(* IEC 61131-3 sources: xPLCCore/codesys_code/Application/COMM_FBs/FB_MpPacker, 25 files *)

(* ---- FB_MpPacker.st ---- *)
FUNCTION_BLOCK FB_MpPacker
VAR_INPUT
END_VAR
VAR_OUTPUT
END_VAR
VAR
    // Builder-pattern slot binding. Caller invokes BindSlot(p) once per
    // reply/event acquisition (TryAcquireReplySlot / ProbeReplySlot /
    // TryAcquireReplySlotOrScratch on AxisGroupSM all auto-bind), then
    // the high-level KV/Pair/Elem helpers below use this stashed pointer
    // instead of taking the slot as a parameter at every call.
    //
    // Default 0 (NULL) -- a Pack* call before BindSlot will deref null
    // and crash deterministically; better than silently writing into
    // a stale slot. Re-bind on every acquire to make stale impossible.
    pSlot : POINTER TO MsgPakInfo := 0;
END_VAR
(* =========== IMPLEMENTATION =========== *)

(* ---- BindSlot.st ---- *)
METHOD BindSlot : BOOL
VAR_INPUT
    pBindSlot : POINTER TO MsgPakInfo;
END_VAR
(* =========== IMPLEMENTATION =========== *)
// Stash the active reply/event slot. All subsequent PackKv* / PackPair*
// / PackElem* / PackKvMap / PackKvArray calls target this slot until
// the next BindSlot. Called automatically by the AxisGroupSM slot-
// lifecycle helpers (TryAcquireReplySlot / ProbeReplySlot /
// TryAcquireReplySlotOrScratch); retry-style sites that hand-roll
// slot acquisition must call this themselves.
pSlot := pBindSlot;
BindSlot := TRUE;

(* ---- PackArrayHeader.st ---- *)
METHOD PackArrayHeader : POINTER TO BYTE
VAR_INPUT
	pStart : POINTER TO BYTE;
	uiCount : UINT;
END_VAR
VAR
	pWordCount : POINTER TO WORD;
END_VAR
(* =========== IMPLEMENTATION =========== *)
// Bound-slot guard (2026-10-04): if pStart lies in the slot bound by
// BindSlot and the up to 3 bytes would not fit, write nothing and flag the
// slot (the post-write checks of the PackKv* helpers only saw the
// overrun after the bytes were already in the next slot).
IF (pSlot <> 0) AND (pStart >= pSlot^.buf) AND (pStart <= pSlot^.buf + pSlot^.buf_capacity) THEN
	IF (pStart - pSlot^.buf) + 3 > TO_DINT(pSlot^.buf_capacity) THEN
		bSlotOverflowed := TRUE;
		pSlot^.overflowed := TRUE;
		PackArrayHeader := pStart;
		RETURN;
	END_IF;
END_IF;
	IF uiCount <= 15 THEN
		pStart^ := 16#90 + UINT_TO_BYTE(uiCount);
		PackArrayHeader := pStart + 1;
	ELSIF uiCount <= 65535 THEN
		pStart^ := 16#DC;
		pStart := pStart + 1;
		pWordCount := pStart;
		Swap16To(ADR(uiCount),pWordCount);
		PackArrayHeader := pStart + 2;
	END_IF;

(* ---- PackBool.st ---- *)
METHOD PackBool : POINTER TO BYTE
VAR_INPUT
	pStart : POINTER TO BYTE;
	bValue : BOOL;
END_VAR
(* =========== IMPLEMENTATION =========== *)
// Bound-slot guard (2026-10-04): if pStart lies in the slot bound by
// BindSlot and the up to 1 bytes would not fit, write nothing and flag the
// slot (the post-write checks of the PackKv* helpers only saw the
// overrun after the bytes were already in the next slot).
IF (pSlot <> 0) AND (pStart >= pSlot^.buf) AND (pStart <= pSlot^.buf + pSlot^.buf_capacity) THEN
	IF (pStart - pSlot^.buf) + 1 > TO_DINT(pSlot^.buf_capacity) THEN
		bSlotOverflowed := TRUE;
		pSlot^.overflowed := TRUE;
		PackBool := pStart;
		RETURN;
	END_IF;
END_IF;
	IF bValue THEN
		pStart^ := 16#C3; // true format
	ELSE
		pStart^ := 16#C2; // false format
	END_IF
	PackBool := pStart + 1;

(* ---- PackDINT.st ---- *)
METHOD PackDINT : POINTER TO BYTE
VAR_INPUT
	pStart : POINTER TO BYTE;
	diValue : DINT;
END_VAR
VAR
	tmpInt : INT;
	pNext : POINTER TO BYTE;
END_VAR
(* =========== IMPLEMENTATION =========== *)
// Bound-slot guard (2026-10-04): if pStart lies in the slot bound by
// BindSlot and the up to 5 bytes would not fit, write nothing and flag the
// slot (the post-write checks of the PackKv* helpers only saw the
// overrun after the bytes were already in the next slot).
IF (pSlot <> 0) AND (pStart >= pSlot^.buf) AND (pStart <= pSlot^.buf + pSlot^.buf_capacity) THEN
	IF (pStart - pSlot^.buf) + 5 > TO_DINT(pSlot^.buf_capacity) THEN
		bSlotOverflowed := TRUE;
		pSlot^.overflowed := TRUE;
		PackDINT := pStart;
		RETURN;
	END_IF;
END_IF;
// Compact signed encoding. Reader already accepts every marker below via
// FB_MpUnpacker.TryReadINT64 / UnpackNext, so shrinking the wire form is a
// pure bandwidth win with no reader-side changes required.

IF diValue >= 0 AND diValue <= 127 THEN
	// positive fixint (0x00-0x7F): 1 byte
	pStart^ := DINT_TO_BYTE(diValue);
	PackDINT := pStart + 1;

ELSIF diValue >= -32 AND diValue < 0 THEN
	// negative fixint (0xE0-0xFF): 1 byte, two's-complement low 8 bits
	pStart^ := DINT_TO_BYTE(diValue);
	PackDINT := pStart + 1;

ELSIF diValue >= -128 AND diValue <= 127 THEN
	// int 8 (0xD0): 2 bytes
	pStart^ := 16#D0;
	pNext := pStart + 1;
	pNext^ := DINT_TO_BYTE(diValue);
	PackDINT := pStart + 2;

ELSIF diValue >= -32768 AND diValue <= 32767 THEN
	// int 16 (0xD1): 3 bytes, big-endian
	pStart^ := 16#D1;
	tmpInt := DINT_TO_INT(diValue);
	Swap16To(ADR(tmpInt), pStart + 1);
	PackDINT := pStart + 3;

ELSE
	// int 32 (0xD2): 5 bytes, big-endian
	pStart^ := 16#D2;
	Swap32To(ADR(diValue), pStart + 1);
	PackDINT := pStart + 5;

END_IF;

(* ---- PackElemDint.st ---- *)
METHOD PackElemDint : BOOL
VAR_INPUT
    diVal : DINT;
END_VAR
(* =========== IMPLEMENTATION =========== *)
// See PackElemStr header. Array-element DINT value, no key, no bump.
pSlot^.whead := PackDINT(pStart := pSlot^.whead, diValue := diVal);
PackElemDint := TRUE;

(* ---- PackElemStr.st ---- *)
METHOD PackElemStr : BOOL
VAR_INPUT
    psVal : POINTER TO STRING;
END_VAR
(* =========== IMPLEMENTATION =========== *)
// Pack one msgpack string value (no key, no count bump). Use INSIDE
// an array body opened by PackKvArray to write one element. The
// outer key + array header (PackKvArray) already counted itself.
pSlot^.whead := PackString(pStart := pSlot^.whead, psValue := psVal);
PackElemStr := TRUE;

(* ---- PackKvArray.st ---- *)
METHOD PackKvArray : BOOL
VAR_INPUT
    psKey    : POINTER TO STRING;
    uiInnerN : UINT;
END_VAR
(* =========== IMPLEMENTATION =========== *)
// Pack one OUTER key + nested-array header into the bound slot, bump
// outer ele_count by 1. Caller follows up with PackElem* calls to fill
// the array. uiInnerN MUST equal the subsequent PackElem* count.
pSlot^.whead := PackString(pStart := pSlot^.whead, psValue := psKey);
pSlot^.whead := PackArrayHeader(pStart := pSlot^.whead, uiCount := uiInnerN);
pSlot^.ele_count := pSlot^.ele_count + 1;
PackKvArray := TRUE;

(* ---- PackKvBool.st ---- *)
METHOD PackKvBool : BOOL
VAR_INPUT
    psKey : POINTER TO STRING;
    bVal  : BOOL;
END_VAR
(* =========== IMPLEMENTATION =========== *)
// See PackKvStr header. KV pair, key:BOOL, bumps outer ele_count by 1.
pSlot^.whead := PackString(pStart := pSlot^.whead, psValue := psKey);
pSlot^.whead := PackBool(pStart := pSlot^.whead, bValue := bVal);
pSlot^.ele_count := pSlot^.ele_count + 1;
PackKvBool := TRUE;

(* ---- PackKvDint.st ---- *)
METHOD PackKvDint : BOOL
VAR_INPUT
    psKey : POINTER TO STRING;
    diVal : DINT;
END_VAR
(* =========== IMPLEMENTATION =========== *)
// See PackKvStr header. KV pair, key:DINT, bumps outer ele_count by 1.
pSlot^.whead := PackString(pStart := pSlot^.whead, psValue := psKey);
pSlot^.whead := PackDINT(pStart := pSlot^.whead, diValue := diVal);
pSlot^.ele_count := pSlot^.ele_count + 1;
PackKvDint := TRUE;

(* ---- PackKvLint.st ---- *)
METHOD PackKvLint : BOOL
VAR_INPUT
    psKey : POINTER TO STRING;
    liVal : LINT;
END_VAR
(* =========== IMPLEMENTATION =========== *)
// See PackKvStr header. KV pair, key:LINT, bumps outer ele_count by 1.
pSlot^.whead := PackString(pStart := pSlot^.whead, psValue := psKey);
pSlot^.whead := PackLINT(pStart := pSlot^.whead, liValue := liVal);
pSlot^.ele_count := pSlot^.ele_count + 1;
PackKvLint := TRUE;

(* ---- PackKvMap.st ---- *)
METHOD PackKvMap : BOOL
VAR_INPUT
    psKey    : POINTER TO STRING;
    uiInnerN : UINT;
END_VAR
(* =========== IMPLEMENTATION =========== *)
// Pack one OUTER key + nested-map header into the bound slot, bump
// outer ele_count by 1. Caller follows up with PackPair* calls to
// fill the inner map. uiInnerN MUST equal the subsequent PackPair*
// count (msgpack readers trust this header, no trailer marker).
pSlot^.whead := PackString(pStart := pSlot^.whead, psValue := psKey);
pSlot^.whead := PackMapHeader(pStart := pSlot^.whead, uiCount := uiInnerN);
pSlot^.ele_count := pSlot^.ele_count + 1;
PackKvMap := TRUE;

(* ---- PackKvReal.st ---- *)
METHOD PackKvReal : BOOL
VAR_INPUT
    psKey : POINTER TO STRING;
    rVal  : REAL;
END_VAR
(* =========== IMPLEMENTATION =========== *)
// See PackKvStr header. KV pair, key:REAL, bumps outer ele_count by 1.
pSlot^.whead := PackString(pStart := pSlot^.whead, psValue := psKey);
pSlot^.whead := PackREAL(pStart := pSlot^.whead, rValue := rVal);
pSlot^.ele_count := pSlot^.ele_count + 1;
PackKvReal := TRUE;

(* ---- PackKvStr.st ---- *)
METHOD PackKvStr : BOOL
VAR_INPUT
    psKey : POINTER TO STRING;
    psVal : POINTER TO STRING;
END_VAR
(* =========== IMPLEMENTATION =========== *)
// Pack one msgpack key:string-value pair into the BOUND slot, bump
// outer ele_count by 1. Slot is set by BindSlot (auto-bound by the
// AxisGroupSM acquire helpers). Pre-2026-06-23 this lived on the
// AxisGroupSM PROGRAM and used an implicit ResponsePacketPointer;
// builder pattern puts msgpack composition where it logically lives
// (the packer) and AxisGroupSM keeps only the slot-lifecycle / FSM
// concerns.
pSlot^.whead := PackString(pStart := pSlot^.whead, psValue := psKey);
pSlot^.whead := PackString(pStart := pSlot^.whead, psValue := psVal);
pSlot^.ele_count := pSlot^.ele_count + 1;
PackKvStr := TRUE;

(* ---- PackLINT.st ---- *)
METHOD PackLINT : POINTER TO BYTE
VAR_INPUT
    pStart  : POINTER TO BYTE;
    liValue : LINT;
END_VAR
VAR
    tmpInt   : INT;
    tmpDint  : DINT;
    pNext    : POINTER TO BYTE;
END_VAR
(* =========== IMPLEMENTATION =========== *)
// Bound-slot guard (2026-10-04): if pStart lies in the slot bound by
// BindSlot and the up to 9 bytes would not fit, write nothing and flag the
// slot (the post-write checks of the PackKv* helpers only saw the
// overrun after the bytes were already in the next slot).
IF (pSlot <> 0) AND (pStart >= pSlot^.buf) AND (pStart <= pSlot^.buf + pSlot^.buf_capacity) THEN
	IF (pStart - pSlot^.buf) + 9 > TO_DINT(pSlot^.buf_capacity) THEN
		bSlotOverflowed := TRUE;
		pSlot^.overflowed := TRUE;
		PackLINT := pStart;
		RETURN;
	END_IF;
END_IF;
// Compact signed encoding (mirrors PackDINT). Wire is interoperable with
// strict MessagePack decoders that reject overlong forms; PLC reader
// accepts every marker via TryReadINT64 / UnpackNext, so shrinking is a
// pure bandwidth win.

IF liValue >= 0 AND liValue <= 127 THEN
    // positive fixint (0x00-0x7F): 1 byte
    pStart^ := DINT_TO_BYTE(LINT_TO_DINT(liValue));
    PackLINT := pStart + 1;

ELSIF liValue >= -32 AND liValue < 0 THEN
    // negative fixint (0xE0-0xFF): 1 byte
    pStart^ := DINT_TO_BYTE(LINT_TO_DINT(liValue));
    PackLINT := pStart + 1;

ELSIF liValue >= -128 AND liValue <= 127 THEN
    // int 8 (0xD0): 2 bytes
    pStart^ := 16#D0;
    pNext := pStart + 1;
    pNext^ := DINT_TO_BYTE(LINT_TO_DINT(liValue));
    PackLINT := pStart + 2;

ELSIF liValue >= -32768 AND liValue <= 32767 THEN
    // int 16 (0xD1): 3 bytes, big-endian
    pStart^ := 16#D1;
    tmpInt := LINT_TO_INT(liValue);
    Swap16To(ADR(tmpInt), pStart + 1);
    PackLINT := pStart + 3;

ELSIF liValue >= -2147483648 AND liValue <= 2147483647 THEN
    // int 32 (0xD2): 5 bytes, big-endian
    pStart^ := 16#D2;
    tmpDint := LINT_TO_DINT(liValue);
    Swap32To(ADR(tmpDint), pStart + 1);
    PackLINT := pStart + 5;

ELSE
    // int 64 (0xD3): 9 bytes, big-endian
    pStart^ := 16#D3;
    Swap64To(ADR(liValue), pStart + 1);
    PackLINT := pStart + 9;

END_IF;

(* ---- PackMapHeader.st ---- *)
METHOD PackMapHeader : POINTER TO BYTE
VAR_INPUT
	pStart : POINTER TO BYTE;
	uiCount : UINT;
	bForceLargeField:BOOL:=FALSE;
END_VAR
VAR
	pWordCount : POINTER TO WORD;
END_VAR
(* =========== IMPLEMENTATION =========== *)
// Bound-slot guard (2026-10-04): if pStart lies in the slot bound by
// BindSlot and the up to 3 bytes would not fit, write nothing and flag the
// slot (the post-write checks of the PackKv* helpers only saw the
// overrun after the bytes were already in the next slot).
IF (pSlot <> 0) AND (pStart >= pSlot^.buf) AND (pStart <= pSlot^.buf + pSlot^.buf_capacity) THEN
	IF (pStart - pSlot^.buf) + 3 > TO_DINT(pSlot^.buf_capacity) THEN
		bSlotOverflowed := TRUE;
		pSlot^.overflowed := TRUE;
		PackMapHeader := pStart;
		RETURN;
	END_IF;
END_IF;
	IF uiCount <= 15 AND bForceLargeField=FALSE THEN
		pStart^ := 16#80 + UINT_TO_BYTE(uiCount);
		PackMapHeader := pStart + 1;
	ELSIF uiCount <= 65535 OR bForceLargeField=TRUE THEN
		pStart^ := 16#DE;
		pStart := pStart + 1;
		pWordCount := pStart;
		Swap16To(ADR(uiCount),pWordCount);
		PackMapHeader := pStart + 2;
	END_IF;

(* ---- PackNil.st ---- *)
METHOD PackNil : POINTER TO BYTE
VAR_INPUT
	pStart : POINTER TO BYTE;
END_VAR
(* =========== IMPLEMENTATION =========== *)
pStart^ := 16#C0; // nil format
PackNil := pStart + 1;

(* ---- PackPairBool.st ---- *)
METHOD PackPairBool : BOOL
VAR_INPUT
    psKey : POINTER TO STRING;
    bVal  : BOOL;
END_VAR
(* =========== IMPLEMENTATION =========== *)
// See PackPairStr header. Nested-map KV, key:BOOL, no outer count bump.
pSlot^.whead := PackString(pStart := pSlot^.whead, psValue := psKey);
pSlot^.whead := PackBool(pStart := pSlot^.whead, bValue := bVal);
PackPairBool := TRUE;

(* ---- PackPairDint.st ---- *)
METHOD PackPairDint : BOOL
VAR_INPUT
    psKey : POINTER TO STRING;
    diVal : DINT;
END_VAR
(* =========== IMPLEMENTATION =========== *)
// See PackPairStr header. Nested-map KV, key:DINT, no outer count bump.
pSlot^.whead := PackString(pStart := pSlot^.whead, psValue := psKey);
pSlot^.whead := PackDINT(pStart := pSlot^.whead, diValue := diVal);
PackPairDint := TRUE;

(* ---- PackPairLint.st ---- *)
METHOD PackPairLint : BOOL
VAR_INPUT
    psKey : POINTER TO STRING;
    liVal : LINT;
END_VAR
(* =========== IMPLEMENTATION =========== *)
// See PackPairStr header. Nested-map KV, key:LINT, no outer count bump.
pSlot^.whead := PackString(pStart := pSlot^.whead, psValue := psKey);
pSlot^.whead := PackLINT(pStart := pSlot^.whead, liValue := liVal);
PackPairLint := TRUE;

(* ---- PackPairReal.st ---- *)
METHOD PackPairReal : BOOL
VAR_INPUT
    psKey : POINTER TO STRING;
    rVal  : REAL;
END_VAR
(* =========== IMPLEMENTATION =========== *)
// See PackPairStr header. Nested-map KV, key:REAL, no outer count bump.
pSlot^.whead := PackString(pStart := pSlot^.whead, psValue := psKey);
pSlot^.whead := PackREAL(pStart := pSlot^.whead, rValue := rVal);
PackPairReal := TRUE;

(* ---- PackPairStr.st ---- *)
METHOD PackPairStr : BOOL
VAR_INPUT
    psKey : POINTER TO STRING;
    psVal : POINTER TO STRING;
END_VAR
(* =========== IMPLEMENTATION =========== *)
// Nested-map KV pair (string value), NO outer ele_count bump.
// Use INSIDE a map opened by PackKvMap -- the outer KvMap counted
// itself; inner pairs are sub-content under that map's header.
pSlot^.whead := PackString(pStart := pSlot^.whead, psValue := psKey);
pSlot^.whead := PackString(pStart := pSlot^.whead, psValue := psVal);
PackPairStr := TRUE;

(* ---- PackREAL.st ---- *)
METHOD PackREAL : POINTER TO BYTE
VAR_INPUT
	pStart : POINTER TO BYTE;
	rValue : REAL;
END_VAR
VAR
	rSwappedValue : REAL;
END_VAR
(* =========== IMPLEMENTATION =========== *)
// Bound-slot guard (2026-10-04): if pStart lies in the slot bound by
// BindSlot and the up to 5 bytes would not fit, write nothing and flag the
// slot (the post-write checks of the PackKv* helpers only saw the
// overrun after the bytes were already in the next slot).
IF pSlot <> 0 THEN	// nested on purpose: ST's AND evaluates every operand (no short circuit)
	IF (pStart >= pSlot^.buf) AND (pStart <= pSlot^.buf + pSlot^.buf_capacity) THEN
		IF (pStart - pSlot^.buf) + 5 > TO_DINT(pSlot^.buf_capacity) THEN
			bSlotOverflowed := TRUE;
			pSlot^.overflowed := TRUE;
			PackREAL := pStart;
			RETURN;
		END_IF;
	END_IF;
END_IF;

    pStart^ := 16#CA;//header for real 32bit
	Swap32To(ADR(rValue),pStart+1);
    PackREAL := pStart + 1+4;

(* ---- PackString.st ---- *)
METHOD PackString : POINTER TO BYTE
VAR_INPUT
	pStart 	: POINTER TO BYTE;
	// --- REVERTED: Input changed back to POINTER TO STRING ---
	// This allows passing ADR('literal') or ADR(variable).
	psValue : POINTER TO STRING;
END_VAR
VAR
	nLen : UDINT;
	pWordLen : POINTER TO WORD;
	// Variables for manual length calculation
	pbyChar : POINTER TO BYTE;
	iLoop   : DINT;

	TMP:WORD;
END_VAR

(* =========== IMPLEMENTATION =========== *)

	// Handle NULL pointer case first
	IF psValue = 0 THEN
		PackString := pStart;
		RETURN;
	END_IF;

	// --- MANUAL LENGTH CALCULATION (USER VALIDATED) ---
	// This loop is essential because LEN(psValue^) may not reflect the true length
	// if the pointer's assumed STRING length is shorter than the actual string.
	nLen := 0;
	pbyChar := psValue; // Get address of the string data from the input pointer
	// Iterate with a large upper bound to ensure null terminator is found,
	// safeguarding against compiler-imposed pointer limits.
	FOR iLoop := 0 TO 999999 DO
	    IF pbyChar^ = 0 THEN // Null terminator found
	        EXIT;
	    END_IF;
	    nLen := nLen + 1;
	    pbyChar := pbyChar + 1;
	END_FOR;
	// -------------------------------------------------

	// Bound-slot guard (2026-10-04): if pStart lies in the slot bound by
	// BindSlot and the header + string bytes would not fit, write nothing and flag the
	// slot (the post-write checks of the PackKv* helpers only saw the
	// overrun after the bytes were already in the next slot).
	IF pSlot <> 0 THEN	// nested on purpose: ST's AND evaluates every operand (no short circuit)
		IF (pStart >= pSlot^.buf) AND (pStart <= pSlot^.buf + pSlot^.buf_capacity) THEN
			IF (pStart - pSlot^.buf) + TO_DINT(nLen) + 3 > TO_DINT(pSlot^.buf_capacity) THEN
				bSlotOverflowed := TRUE;
				pSlot^.overflowed := TRUE;
				PackString := pStart;
				RETURN;
			END_IF;
		END_IF;
	END_IF;
	IF nLen <= 31 THEN
		pStart^ := 16#A0 + UDINT_TO_BYTE(nLen);
		pStart := pStart + 1;
	ELSIF nLen <= 255 THEN
		pStart^ := 16#D9;
		pStart := pStart + 1;
		pStart^ := UDINT_TO_BYTE(nLen);
		pStart := pStart + 1;
	ELSIF nLen <= 65535 THEN
		pStart^ := 16#DA;
		pStart := pStart + 1;
		pWordLen := pStart;
		//pWordLen^ := SwapWORD(UDINT_TO_WORD(nLen));

		TMP:=UDINT_TO_WORD(nLen);
		Swap16To(ADR(TMP),pWordLen);
		pStart := pStart + 2;
	ELSE
		PackString := pStart; // String is too long for MessagePack formats
		RETURN;
	END_IF;

	// Copy string data using the original input pointer
	MEMUtils.MemCpy(pbyDest:=pStart, pbySrc:=psValue, dwSize:=UDINT_TO_DWORD(nLen));
	PackString := pStart + nLen;

(* ---- SwapREAL.st ---- *)
(*
Helper method for swapping byte order for REAL (Little-Endian to Big-Endian)
*)
METHOD PRIVATE SwapREAL : REAL
VAR_INPUT
	rValue : REAL;
END_VAR
VAR
	rSwapped : REAL;
	prIn : POINTER TO ARRAY[0..3] OF BYTE;
	prOut : POINTER TO ARRAY[0..3] OF BYTE;
END_VAR
(* =========== IMPLEMENTATION =========== *)
	prIn := ADR(rValue);
	prOut := ADR(rSwapped);
	prOut^[0] := prIn^[3];
	prOut^[1] := prIn^[2];
	prOut^[2] := prIn^[1];
	prOut^[3] := prIn^[0];
	SwapREAL := rSwapped;
